FUNCTION_BLOCK FB_FeedMeina2_500x500_Circles EXTENDS FB_RecipeBase

METHOD Build : BOOL
VAR
    TotalX, TotalY             : LREAL;
    CircleRadius               : LREAL;
    Velo                       : LREAL;
    localConfig                : ST_GantryXYZ_Config;
    
    X_Offset                   : LREAL; 
    Y_Offset                   : LREAL;
    p                          : INT;

    PanelW                     : ARRAY[1..10] OF LREAL; 
    PanelH                     : ARRAY[1..10] OF LREAL; 
    PanelX                     : ARRAY[1..10] OF LREAL; 
    PanelY                     : ARRAY[1..10] OF LREAL; 

    HoleDistanceFromEdgeOfRail : LREAL := 100.0;
    SomeFixedDimension         : LREAL := 12.63;
    PanelRailOffsetX           : LREAL;
    PanelRailOffsetY           : LREAL;
    ExtrusionLengthX           : LREAL;
    ExtrusionLengthY           : LREAL;
    BaseExtrusion              : LREAL; 
    
    NumberOfHolesX             : INT := 3;
    NumberOfHolesY             : INT := 5;
    HolesSpacingX              : LREAL;
    HolesSpacingY              : LREAL;
    
    i                          : INT;
    holeIdx                    : INT;
    
    RailSlot                   : LREAL := 29.0;
    BigSlot                    : LREAL := 200.0;
    SmallSlot                  : LREAL := 100.0;

    LeadInY                    : LREAL := 10.0;
    LeadOutY                   : LREAL := 10.0;

    sx                         : LREAL;
    sy                         : LREAL;
    dx                         : LREAL;
    dy                         : LREAL;
    r_val                      : LREAL;
END_VAR
_Busy := TRUE;
_Done := FALSE;
_Error := FALSE;
Build := FALSE;
THIS^.UpdateNestingLimits();

IF NOT _Config.IsValid THEN
    _Busy := FALSE;
    _Error := TRUE; 
    Build := FALSE;
    RETURN;
END_IF

PanelX[1] := 0.0;            PanelY[1] := 0.0;
PanelW[1] := 1000.0;         PanelH[1] := 1000.0;
_ShapeStart[1].X := PanelX[1] + PanelW[1];
_ShapeStart[1].Y := PanelY[1] + (PanelH[1] / 2.0) - LeadInY;

PanelX[2] := 0.0;            PanelY[2] := 1020.0;
PanelW[2] := 500.0;          PanelH[2] := 500.0;
_ShapeStart[2].X := PanelX[2] + PanelW[2];
_ShapeStart[2].Y := PanelY[2] + (PanelH[2] / 2.0) - LeadInY;

PanelX[3] := 0.0;            PanelY[3] := 1540.0;
PanelW[3] := 500.0;          PanelH[3] := 500.0;
_ShapeStart[3].X := PanelX[3] + PanelW[3];
_ShapeStart[3].Y := PanelY[3] + (PanelH[3] / 2.0) - LeadInY;

PanelX[4] := 520.0;          PanelY[4] := 1020.0;
PanelW[4] := 500.0;          PanelH[4] := 500.0;
_ShapeStart[4].X := PanelX[4] + PanelW[4];
_ShapeStart[4].Y := PanelY[4] + (PanelH[4] / 2.0) - LeadInY;

PanelX[5] := 520.0;          PanelY[5] := 1540.0;
PanelW[5] := 500.0;          PanelH[5] := 500.0;
_ShapeStart[5].X := PanelX[5] + PanelW[5];
_ShapeStart[5].Y := PanelY[5] + (PanelH[5] / 2.0) - LeadInY;

holeIdx := 0; 

FOR p := 1 TO 5 DO
    TotalX := PanelW[p];
    TotalY := PanelH[p];
    X_Offset := PanelX[p];
    Y_Offset := PanelY[p];

    PanelRailOffsetX := 0.1 * TotalX;
    PanelRailOffsetY := 0.1 * TotalY;

    ExtrusionLengthX := TotalX - (2.0 * PanelRailOffsetX);
    ExtrusionLengthY := TotalY - (2.0 * PanelRailOffsetY);

    IF NumberOfHolesX > 1 THEN
        HolesSpacingX := (ExtrusionLengthX - (2.0 * HoleDistanceFromEdgeOfRail)) / INT_TO_LREAL(NumberOfHolesX - 1);
    ELSE
        HolesSpacingX := 0.0;
    END_IF

    IF NumberOfHolesY > 1 THEN
        HolesSpacingY := (ExtrusionLengthY - (2.0 * HoleDistanceFromEdgeOfRail)) / INT_TO_LREAL(NumberOfHolesY - 1);
    ELSE
        HolesSpacingY := 0.0;
    END_IF

    holeIdx := holeIdx + 1;
    _HolesDrill[holeIdx].X := LREAL_TO_REAL((TotalX / 2.0) + X_Offset);
    _HolesDrill[holeIdx].Y := LREAL_TO_REAL((TotalY / 2.0) + Y_Offset);

    FOR i := NumberOfHolesY TO 1 BY -1 DO
        holeIdx := holeIdx + 1;
        _HolesDrill[holeIdx].X := LREAL_TO_REAL(PanelRailOffsetX - SomeFixedDimension + X_Offset);
        _HolesDrill[holeIdx].Y := LREAL_TO_REAL(PanelRailOffsetY + HoleDistanceFromEdgeOfRail + ((i - 1) * HolesSpacingY) + Y_Offset);
    END_FOR

    FOR i := 1 TO NumberOfHolesX DO
        holeIdx := holeIdx + 1;
        _HolesDrill[holeIdx].X := LREAL_TO_REAL(PanelRailOffsetX + HoleDistanceFromEdgeOfRail + ((i - 1) * HolesSpacingX) + X_Offset);
        _HolesDrill[holeIdx].Y := LREAL_TO_REAL(PanelRailOffsetY - SomeFixedDimension + Y_Offset);
    END_FOR

    FOR i := 1 TO NumberOfHolesY DO
        holeIdx := holeIdx + 1;
        _HolesDrill[holeIdx].X := LREAL_TO_REAL(PanelRailOffsetX + ExtrusionLengthX + SomeFixedDimension + X_Offset);
        _HolesDrill[holeIdx].Y := LREAL_TO_REAL(PanelRailOffsetY + HoleDistanceFromEdgeOfRail + ((i - 1) * HolesSpacingY) + Y_Offset);
    END_FOR

    FOR i := NumberOfHolesX TO 1 BY -1 DO
        holeIdx := holeIdx + 1;
        _HolesDrill[holeIdx].X := LREAL_TO_REAL(PanelRailOffsetX + HoleDistanceFromEdgeOfRail + ((i - 1) * HolesSpacingX) + X_Offset);
        _HolesDrill[holeIdx].Y := LREAL_TO_REAL(PanelRailOffsetY + ExtrusionLengthY + SomeFixedDimension + Y_Offset);
    END_FOR
END_FOR

_HolesToDrill := holeIdx;

_ShapesCount := 10; 

_ShapeStart[6].X := 1030.0; _ShapeStart[6].Y := 0.0;
_ShapeStart[7].X := 1090.0; _ShapeStart[7].Y := 0.0;
_ShapeStart[8].X := 210.0;  _ShapeStart[8].Y := 2200.0;
_ShapeStart[9].X := 410.0;  _ShapeStart[9].Y := 2150.0;
_ShapeStart[10].X := 810.0; _ShapeStart[10].Y := 2150.0;

IF _ConfigProvider <> 0 THEN
    localConfig := _ConfigProvider.Config;
    Velo := localConfig.CuttingSpeedXY;
ELSE
    Velo := 50.0;
END_IF

_GeometryWriter.Clear();
_GeometryWriter.EnableTangentialFollowing();

sx := 0.0; sy := 0.0; dx := 0.0; dy := 0.0; r_val := 0.0;

CASE _CurrentShapeIndex OF
    1, 2, 3, 4, 5:
        sx := PanelX[_CurrentShapeIndex];
        sy := PanelY[_CurrentShapeIndex];
        TotalX := PanelW[_CurrentShapeIndex];
        TotalY := PanelH[_CurrentShapeIndex];
        CircleRadius := TotalX / 2.0;

        _GeometryWriter.AddStartPoint(_ShapeStart[_CurrentShapeIndex].X, _ShapeStart[_CurrentShapeIndex].Y); 
        
        _GeometryWriter.AddLine(sx + TotalX, sy + CircleRadius, Velo); 
        
        _GeometryWriter.AddArc(sx, sy + CircleRadius, sx + CircleRadius, sy + CircleRadius, Velo, FALSE);
        
        _GeometryWriter.AddArc(sx + TotalX, sy + CircleRadius, sx + CircleRadius, sy + CircleRadius, Velo, FALSE);
        
        _GeometryWriter.AddLine(sx + TotalX, sy + CircleRadius + LeadOutY, Velo); 

    6, 7, 8, 9, 10:
        sx := _ShapeStart[_CurrentShapeIndex].X;
        sy := _ShapeStart[_CurrentShapeIndex].Y;
        r_val := 10.0;

        BaseExtrusion := 800.0; 

        IF _CurrentShapeIndex = 6 THEN
            dx := RailSlot;
            dy := BaseExtrusion;
        ELSIF _CurrentShapeIndex = 7 THEN
            dx := RailSlot;
            dy := BaseExtrusion; 
        ELSIF _CurrentShapeIndex = 8 THEN
            dx := SmallSlot;
            dy := SmallSlot;
        ELSIF _CurrentShapeIndex = 9 THEN
            dx := BigSlot;
            dy := BigSlot;
        ELSIF _CurrentShapeIndex = 10 THEN
            dx := BigSlot;
            dy := BigSlot;
        END_IF

        _GeometryWriter.AddStartPoint(sx, sy);

        _GeometryWriter.AddLine(sx, sy + dy - r_val, Velo);
        IF r_val > 0 THEN
            _GeometryWriter.AddArc(sx + r_val, sy + dy, sx + r_val, sy + dy - r_val, Velo, TRUE);
        END_IF

        _GeometryWriter.AddLine(sx + dx - r_val, sy + dy, Velo);
        IF r_val > 0 THEN
            _GeometryWriter.AddArc(sx + dx, sy + dy - r_val, sx + dx - r_val, sy + dy - r_val, Velo, TRUE);
        END_IF

        _GeometryWriter.AddLine(sx + dx, sy + r_val, Velo);
        IF r_val > 0 THEN
            _GeometryWriter.AddArc(sx + dx - r_val, sy, sx + dx - r_val, sy + r_val, Velo, TRUE);
        END_IF

        _GeometryWriter.AddLine(sx + r_val, sy, Velo);
        IF r_val > 0 THEN
            _GeometryWriter.AddArc(sx, sy + r_val, sx + r_val, sy + r_val, Velo, TRUE);
        END_IF

END_CASE

_GeometryWriter.EndTable();

_Busy := FALSE;
_Done := TRUE;
Build := TRUE;
END_METHOD

METHOD PROTECTED CalculateFootprint
VAR_INPUT
END_VAR
_NominalX := 1200;
_NominalY := 2400;
END_METHOD

PROPERTY ExecutionRoute : E_ExecutionRoute
GET
ExecutionRoute := E_ExecutionRoute.eFeedTable;
END_GET
END_PROPERTY

METHOD FB_init : BOOL
VAR_INPUT
	bInitRetains : BOOL; // if TRUE, the retain variables are initialized (warm start / cold start)
	bInCopyCode : BOOL;  // if TRUE, the instance afterwards gets moved into the copy code (online change)
END_VAR
_Limits.PanelFrontLength.MinVal := 100.0;
_Limits.PanelFrontLength.MaxVal := 2400.0;

_Limits.PanelFrontWidth.MinVal  := 100.0;
_Limits.PanelFrontWidth.MaxVal  := 1200.0;

_Limits.PanelHeight.MinVal      := 0.0;
_Limits.PanelHeight.MaxVal      := 0.0;

_Limits.RailHeightCorrection.MinVal := 0.0;
_Limits.RailHeightCorrection.MaxVal := 0.0;

_Limits.CuttingOverpass.MinVal := 0.0;
_Limits.CuttingOverpass.MaxVal := 50.0;

_Limits.GroovingOverpass.MinVal := 0.0;
_Limits.GroovingOverpass.MaxVal := 50.0;

_Limits.GrooveDepthZ.MinVal := 0.0;
_Limits.GrooveDepthZ.MaxVal := 9.0; 

_Limits.CuttingOverpass.MinVal := 0.0;
_Limits.CuttingOverpass.MaxVal := 50.0;
_Limits.GroovingOverpass.MinVal := 0.0;
_Limits.GroovingOverpass.MaxVal := 50.0;

_Limits.Radius.MinVal := 10.0;     
_Limits.Radius.MaxVal := 600.0;
END_METHOD

END_FUNCTION_BLOCK

(* stored: Version 1.1.0.1, ProductVersion 3.1.4024.15
   POU FB_FeedMeina2_500x500_Circles: Id {c6c41331-3824-483b-a50b-8cfea9f566ab}, SpecialFunc None
   Method Build: Id {5627da5e-3b90-4d43-82c7-27af2973971b}
   Method CalculateFootprint: Id {b7a26e0e-4a5c-4d2c-b3fb-2dac1886af28}
   Property ExecutionRoute: Id {71a08135-19bd-49fc-aa74-ad4fd8d9fa3a}
   Get Get: Id {799a229d-23d2-4133-8efe-eaedb6d63500}
   Method FB_init: Id {d1276162-3835-4b38-af75-eceb704f22ca} *)
